// 	3: stStationPoses.aPoseLargeMotorPickupSt1 := stStation.stSts3.aPoseLargeMotorPickupSt1;
// 		stStationPoses.aPoseLargeMotorPickupSt2 := stStation.stSts3.aPoseLargeMotorPickupSt2;
// 		stStationPoses.aPoseLargeMotorPickupSt3 := stStation.stSts3.aPoseLargeMotorPickupSt3;
// 		stStationPoses.aPoseLargeMotorPlaceSt1 := stStation.stSts3.aPoseLargeMotorPlaceSt1;
// 		stStationPoses.aPoseLargeMotorPlaceSt2 := stStation.stSts3.aPoseLargeMotorPlaceSt2;
// 		stStationPoses.aPoseLargeMotorPlaceSt3 := stStation.stSts3.aPoseLargeMotorPlaceSt3;
// 		stStationPoses.aPoseMirrorAdj := stStation.stSts3.aPoseMirrorAdj;
// 		stStationPoses.aPoseMirrorPickupSt1 := stStation.stSts3.aPoseMirrorPickupSt1;
// 		stStationPoses.aPoseMirrorPickupSt2 := stStation.stSts3.aPoseMirrorPickupSt2;
// 		stStationPoses.aPoseMirrorPlaceSt1 := stStation.stSts3.aPoseMirrorPlaceSt1;
// 		stStationPoses.aPoseMirrorPlaceSt2 := stStation.stSts3.aPoseMirrorPlaceSt2;
// 		stStationPoses.aPoseMirrorPlaceSt3 := stStation.stSts3.aPoseMirrorPlaceSt3;
// 		stStationPoses.aPoseSmallMotorPlaceSt1 := stStation.stSts3.aPoseSmallMotorPlaceSt1;
// 		stStationPoses.aPoseSmallMotorPlaceSt2 := stStation.stSts3.aPoseSmallMotorPlaceSt2;
// 		stStationPoses.aPoseSmallMotorPickupSt1 := stStation.stSts3.aPoseSmallMotorPickupSt1;
// 		stStationPoses.aPoseSmallMotorPickupSt2 := stStation.stSts3.aPoseSmallMotorPickupSt2;
// 		stStationPoses.aPoseSmallMotorPickupSt3 := stStation.stSts3.aPoseSmallMotorPickupSt3;
// 		stStationPoses.aPosePassedLargeSt1 := stStation.stSts3.aPosePassedLargeSt1;
// 		stStationPoses.aPosePassedLargeSt2 := stStation.stSts3.aPosePassedLargeSt2;
// 		stStationPoses.aPosePassedLargeSt3 := stStation.stSts3.aPosePassedLargeSt3;
// 		stStationPoses.aPosePassedSmallSt1 := stStation.stSts3.aPosePassedSmallSt1;
// 		stStationPoses.aPosePassedSmallSt2 := stStation.stSts3.aPosePassedSmallSt2;
// 		stStationPoses.aPosePassedSmallSt3 := stStation.stSts3.aPosePassedSmallSt3;
// 		stStationPoses.aPosePassedSmallSt4 := stStation.stSts3.aPosePassedSmallSt4;
// 		stStationPoses.rLinPosPalletPass := stStation.stSts3.rLinPosPalletPass;
// 		stStationPoses.rLinPosPalletReject := stStation.stSts3.rLinPosPalletReject;
// 		stStationPoses.rLinPosMotorPickup := stStation.stSts3.rLinPosMotorPickup;
// 		stStationPoses.rLinPosMirrorPickup := stStation.stSts3.rLinPosMirrorPickup;
// 		stStationPoses.rLinPosPlace := stStation.stSts3.rLinPosPlace;
END_CASE
END_METHOD

END_FUNCTION_BLOCK

(* stored: Version 1.1.0.1
   POU FB_Operating: Id {cb20d2d7-f855-4aae-b705-a3965881f189}, SpecialFunc None
   Folder Act: Id {fbbec362-08eb-40d4-b222-e2740caef989}
   Folder Mth: Id {417f24a5-3b5e-420c-a919-64423eab2c88}
   Method AdjDone: Id {ccf00eb9-e52d-4e13-9f7e-5744fa517659}
   Method CheckProduct: Id {04076697-36a3-4c55-b410-5e8547b43894}
   Method CheckType: Id {8d7e3152-2bba-40d1-9708-3b600a5e1cec}
   Method DisableSetStation: Id {1df013af-16bc-43b7-90ef-e92dda3557f5}
   Method DismountingDone: Id {a39cabe4-9e85-4206-a432-3eb78aadc624}
   Method EngageHolder: Id {2124621f-833e-4b2e-bd6d-347e3d6cfabe}
   Method EngageSlider: Id {8e1fe543-8a53-46fd-8dd7-5f5324a72a63}
   Action Finished14mm: Id {90d4519f-ee19-45e8-93b6-61a6b2f8595a}
   Action Galvo10mm: Id {28526a0e-eb6d-4d21-9b51-86ca0eddfaa9}
   Action Galvo14mm: Id {6b89f09a-61d6-4595-b012-fc055ca97ffe}
   Method Initialize: Id {b1d364bc-92df-4ed4-bb2e-dbdc6cd8f730}
   Action MirrorAdj: Id {d13ff194-9dff-4689-a5fd-bbb4b7d4855a}
   Method MirrorOffset: Id {f2318cd9-c83e-421e-8ac9-a9145489dd90}
   Method ReleaseHolder: Id {fced77fd-576b-4edd-aadf-26a3e3edd780}
   Method ReleaseSlider: Id {23f91438-bd72-42e7-b6f5-3d7640c0ab5c}
   Method SetAdjustmentPoses: Id {075017d8-2792-4614-9697-ca6eae04e726}
   Method WritePoses: Id {6a3f8326-bb08-4c0f-baff-34c018bd39d1} *)
